(* Logix 5000 project; controller Transcat_L33ER vendor 1 type 14 code 107 rev 32.11; software revision 32.02 *)
// Upgraded CPLX to handle up to 32 EIP Nodes

TASK MainTask (continuous, watchdog 500 ms) : MainProgram

MODULES
   Local : vendor 1 type 14 code 107 (Compact 0, rev 32.11)
        TC_Remote_IO:5:O.0   // HOIST 2 BEACON RED
        TC_Remote_IO:5:O.1   // CV_101 - 3 Way Valve - Recyle / Process
        TC_Remote_IO:3:O.6   // HOIST 1 Beacon Red
        TC_Remote_IO:3:O.5   // HOIST 1 BEACON GREEN
        TC_Remote_IO:3:O.7   // Hoist 2 BEACON GREEN
        TC_Remote_IO:3:O   // HOIST 1 RED
      VFD9_Screener : PowerFlex 525-EENET (Ethernet 192.168.1.199, rev 5.1, Output RPI 20 ms)   // Screener Kaison
      GF201_Bentonite_Feeder : PowerFlex 525-EENET (Ethernet 192.168.1.195, rev 5.1, Output RPI 20 ms)   // Thayer Weigh Belt Feeder
      MX101_UpperHowesVFD : PowerFlex 525-EENET (Ethernet 192.168.1.191, rev 5.1, Output RPI 20 ms)   // VFD for Upper Howes Mixer
           MX101_UpperHowesVFD:I.Ready   // UpperHowes Drive Ready Status
           MX101_UpperHowesVFD:I.DriveStatus.1   // 1 = Running, 0 - Stopped
           MX101_UpperHowesVFD:I.DriveStatus.0   // 1 = Drive is Ready
           MX101_UpperHowesVFD:I.DriveStatus.4   // 1 = Accelerating
           MX101_UpperHowesVFD:I.DriveStatus.10   // 1 - parameter locked
           MX101_UpperHowesVFD:I.DriveStatus.8   // 1 = At Referecne Speed
           MX101_UpperHowesVFD:I.Faulted   // UpperHowes Drive Faulted
           MX101_UpperHowesVFD:I.DriveStatus.6   // not used
           MX101_UpperHowesVFD:I.DriveStatus.9   // 1 - Main Freq by Active Comms
           MX101_UpperHowesVFD:I.DriveStatus.3   // 1 = Rotating Forward
           MX101_UpperHowesVFD:I.DriveStatus.7   // 1= Faulted
           MX101_UpperHowesVFD:I.DriveStatus.2   // 1 = Forward, 0 = Reverse
           MX101_UpperHowesVFD:I.Active   // UpperHowes Drive Active
           MX101_UpperHowesVFD:I.DriveStatus.5   // 1= Decelerating
           MX101_UpperHowesVFD:O.Start   // Drive Start
           MX101_UpperHowesVFD:O.FreqCommand   // Input Hz into Source A: 0-60 Hz range
           MX101_UpperHowesVFD:O.Stop   // Drive Stop
      VF101_Medium_Feeder : PowerFlex 525-EENET (Ethernet 192.168.1.196, rev 5.1, Output RPI 20 ms)   // Medium Feeder
      MX201_LowerHowesVFD : PowerFlex 525-EENET (Ethernet 192.168.1.192, rev 5.1, Output RPI 20 ms)   // VFD for Lower Howes Mixer
           MX201_LowerHowesVFD:I.Ready   // LowerHowes Drive Ready Status
           MX201_LowerHowesVFD:I.Faulted   // LowerHowes Drive Faulted
           MX201_LowerHowesVFD:I.Active   // LowerHowes Drive Active
           MX201_LowerHowesVFD:O.Stop   // Drive Stop
      VF201_Small_Feeder_2 : PowerFlex 525-EENET (Ethernet 192.168.1.197, rev 5.1, Output RPI 20 ms)   // Acrison Small Feeder 2
      Anybus_ETH_SER : ETHERNET-MODULE (Ethernet 192.168.1.127, rev 1.1, Output RPI 50 ms)   // Anybus gateway from serial (Bronkhorst) to / from EIP (Ether/IP) - PLC
      SBC2000_1_Acrison : ETHERNET-MODULE (Ethernet 192.168.1.150, rev 1.1, Output RPI 250 ms)   // Acrison Drive 1 to control Small Feeder 1
           SBC2000_1_Acrison:I.Data   // Ethernet Input Array
           SBC2000_1_Acrison:I.Data[1]   // PV - Feedrate - kg/hr
           SBC2000_1_Acrison:I.Data[2]   // Totalizer 1 - kg
           SBC2000_1_Acrison:I.Data[4]   // Hopper Level - %
           SBC2000_1_Acrison:I.Data[0]   // SP-FeedRate - kg/hr
           SBC2000_1_Acrison:I.Data[3]   // OT - Motor Speed - %
           SBC2000_1_Acrison:O.Data[15]   // When Command_Bits is 1, machine is running.
      Thayer1_BS : ETHERNET-MODULE (Ethernet 192.168.1.140, rev 1.1, Output RPI 50 ms)   // Thayer 1 Weight Belt Feeder
      Thayer2_BS : ETHERNET-MODULE (Ethernet 192.168.1.160, rev 1.1, Output RPI 50 ms)   // Thayer 2 Weigh Belt Feeder
      XS26_VFD_Cabinet_Safety_Controller : XS26 SC26 SC10 (Ethernet 192.168.1.212, rev 2.1, StandardDataDriven RPI 100 ms)   // Banner XS26 Safety Controller with 3 expansion modules in VFD cabinet
           XS26_VFD_Cabinet_Safety_Controller:I1.Data[0].7   // MX101 VFD STO - OK
           XS26_VFD_Cabinet_Safety_Controller:I1.Data[1].0   // MX201 VFD STO - OK
      XS26_PLC_Safety_Controller : XS26 SC26 SC10 (Ethernet 192.168.1.211, rev 2.1, StandardDataDriven RPI 100 ms)   // XS26 Safety Controller in PLC cabinet
      TC_Remote_IO : 1734-AENT (Ethernet 192.168.1.190, rev 6.1, Output RPI 20 ms)
         TC_8Pt_Analog_Input : vendor 1 type 115 code 210 (PointIO 1, rev 3.1, Input RPI 80 ms)
         TC_8pt_DC_Input_Sink : 1734-IB8 (PointIO 2, rev 3.1)
         TC_8pt_Digital_Output_Sourced : 1734-OB8 (PointIO 3, rev 3.1)
          : 1734-OB8 (PointIO 5, rev 3.1)   // For Hoist Safety Beacon
         TC_4pt_Relay_Output : 1734-OW4 (PointIO 4, rev 3.1)
END_MODULES

TYPE Acrison_Feeder :   // Acrison Feeder Tags
STRUCT
   AutoMan : BOOL;   // On - Auto Control - follows AutoRun bit, Off - Manaul Control - follows Manual Run bit
   ManualRun : BOOL;   // On - Runs feeder in Manual, Off - Stops feeder in manual
   AutoRun : BOOL;   // On - Runs feeder in Auto Off - Stops feeder in Auto
   Interlock : BOOL;   // Interlock bit - if on - Feeder will not run
   Output : BOOL;   // On - Feeder runs, Off Feeder stops
   Int_Status : DINT;   // 32 Status bits from feeder
   SP_HMI : REAL;   // setpoint from HMI
   SP_READ : REAL;   // setpoint read back from controller
   Enable : BOOL;   // Enable logic to run feeder
   OT_Actual_Hz : REAL;   // The current output of the VFD in Hz
   FreqHz_Real : REAL;   // The command frequency of the drive in Hz
   CycleTime : TIMER;   // running time of current cycle
   CampTime : TIMER;   // running time of current campaign / batch
   TotalTime : TIMER;   // total time the device / motor has run since last reset
   OneShots : BOOL[32];   // 32 Booleans to hold one-shots assicated with this device
   TimeRunTarget : DINT;   // Target Amount of time in seconds to run the device
   StartDelay : TIMER;   // Delay before motor start
   StartDelayms : DINT;   // Start delay in milliseconds
   TimeRunStart : BOOL;   // Bit to start and run a timed run
   RPM : REAL;   // RPM of shaft
END_STRUCT
END_TYPE

TYPE BronkhorstFlowMeter :   // Read and write values for Bronkhorst Flow Meters
STRUCT
   SP_R : REAL;   // Set Point - FlowRate - Read - g/min - read from Flow Meter
   PV_R : REAL;   // Process Variable - FlowRate - Read - g/min
   OT_R : REAL;   // Output - PumpSpeed - Read - %
   TempC : REAL;   // Temperaure - Read - Deg C
   Density : REAL;   // Density - Read - g/liter
   Usertag : STRING;   // User Tag in Flow Meter - String
   FBNode : INT;   // Flow Bus Node # - Integer
   Model : STRING;   // Flow Meter Model #
   Serial : STRING;   // Flow Meter Serial #
   Capacity : REAL;   // Max Flow Rate of Flow Meter
   Enable : BOOL;   // Device enable bit
   AutoMan : BOOL;   // Select Auto / Manual Mode
   AutoRun : BOOL;   // On / Off in Auto Mode
   ManualRun : BOOL;   // On / Off- in Manual Mode
   Interlock : BOOL;   // Interlock Bit
   Output : BOOL;   // Output Bit for Device
   SP_HMI : REAL;   // Setpoint from HMI
   SP_W : REAL;   // Setpoint - flowrate g/min - write to Flow Meter from PLC
   Connected : BOOL;   // Is flow meter connecte to the flow bus network
   Alarm : BOOL;   // Alarm Bit - if on flow meter in ALarm Status
   Running : BOOL;   // the flow meter is running / dosing
   AlarmReset : BOOL;   // bit to toggle to reset alarm
   AlarmID : INT;   // Integer # that describes the type of Alarm
   ReadTime : INT;   // time in milliseconds to read the flow meter data
   DevPct : REAL;   // % deviation of process variable from setpoint
   CycleTime : TIMER;   // running time of current cycle
   CampTime : TIMER;   // running time of current campaign
   TotalTime : TIMER;   // total time the device / motor has run since last reset
   OneShots : BOOL[32];   // 32 Booleans to hold one-shots assicated with this device
   TimeRunTarget : DINT;   // Target Amount of time in seconds to run the device
   StartDelay : TIMER;   // Delay before motor start
   StartDelayms : DINT;   // Start delay in milliseconds
   TimeRunStart : BOOL;   // Bit to start and run a timed run
   Totalizer : REAL;   // Total dosed by flow meter since last reset
   TotalizerReset : BOOL;   // Bit to reset the totalizer (called a counter in Bronkhorst literature)
   TotalizerEnable : BOOL;   // Bit to turn the totalizer on / off
   HighPressureLimit_HMI : REAL;   // High Pressure Limit Real Value in psi from HMI
   HighPressureLimit_Int : DINT;   // High Pressure limit converted to Int * 100 so 40.0 real = 4000 Int value
   HighPressureTime : DINT;   // Presistance time for high pressure limit
   HighPressureTimer : TIMER;   // Timer to time how many consecutive seconds the line pressur can stay above the limit before interlockig the pump / flow meter system
   HighPressureInterlock : BOOL;   // The pump / flow meter dosign system is interlocked due to a high pressure event
   TotalResetCmd : BOOL;   // Total Reset Command from HMI
   TotalResetDone : BOOL;   // Gateway confirms totalizer is near zero
   TotalResetError : BOOL;   // Reset failed after the retry limit
   AlarmResetCmd : BOOL;   // PLC/HMI requests alarm reset
   AlarmResetDone : BOOL;   // Gateway confirms alarm reset
   AlarmResetError : BOOL;   // Alarm didn't clear / reset failed
   TotalResetAttempts : DINT;   // Total Reset Attempts
   CommOK : BOOL;   // Meter communications are healthy
   DataValid : BOOL;   // Current data is good and not stale
   DataStale : BOOL;   // Data is no longer considered current
   DataAgeMs : DINT;   // Milliseconds since last good meter data
END_STRUCT
END_TYPE

TYPE Device :   // this UDT will be the template for all equipment / devices - feeders, flow meters, others and will be set up for each device to be indexed and processed via indirect addressing
STRUCT
   SP_R : REAL;   // Set Point - FlowRate - Read - g/min - read from Flow Meter
   PV_R : REAL;   // Process Variable - FlowRate - Read - g/min
   OT_R : REAL;   // Output - PumpSpeed - Read - %
   TempC : REAL;   // Temperaure - Read - Deg C
   Density : REAL;   // Density - Read - g/liter
   Usertag : STRING;   // User Tag in Flow Meter - String
   FBNode : INT;   // Flow Bus Node # - Integer
   Model : STRING;   // Flow Meter Model #
   Serial : STRING;   // Flow Meter Serial #
   Capacity : REAL;   // Max Flow Rate of Flow Meter
   Enable : BOOL;   // Device enable bit
   AutoMan : BOOL;   // Select Auto / Manual Mode
   AutoRun : BOOL;   // On / Off in Auto Mode
   ManualRun : BOOL;   // On / Off- in Manual Mode
   Interlock : BOOL;   // Interlock Bit
   Output : BOOL;   // Output Bit for Device
   SP_HMI : REAL;   // Setpoint from HMI
   SP_W : REAL;   // Setpoint - flowrate g/min - write to Flow Meter from PLC
   Connected : BOOL;   // Is flow meter connecte to the flow bus network
   Alarm : BOOL;   // Alarm Bit - if on flow meter in ALarm Status
   Running : BOOL;   // the flow meter is running / dosing
   AlarmReset : BOOL;   // bit to toggle to reset alarm
   AlarmID : INT;   // Integer # that describes the type of Alarm
   ReadTime : INT;   // time in milliseconds to read the flow meter data
   DevPct : REAL;   // % deviation of process variable from setpoint
   CycleTime : TIMER;   // running time of current cycle
   CampTime : TIMER;   // running time of current campaign
   TotalTime : TIMER;   // total time the device / motor has run since last reset
   OneShots : BOOL[32];   // 32 Booleans to hold one-shots assicated with this device
   TimedRunTarget : DINT;   // Target Amount of time in seconds to run the device
   StartDelay : TIMER;   // Delay before motor start
   StartDelayms : DINT;   // Start delay in milliseconds
   TimeRunEnable : BOOL;   // Bit to enable / activate a timed (campaign timed) run
   Totalizer : REAL;   // Total dosed by flow meter since last reset
   TotalizerReset : BOOL;   // Bit to reset the totalizer (called a counter in Bronkhorst literature)
   TotalizerEnable : BOOL;   // Bit to turn the totalizer on / off
   TimedRunTargetms : DINT;   // Timed run target convered to ms for use in timers
   OutPutTest : BOOL;   // A bit to simulate output that does NOT control anything
   StartDelay_ST_Timer : FBD_TIMER;   // Start delay timer to use in stuctured text
   PermissivesAuto : BOOL;   // Bit to allow device to start in AUTO as long as all permissive conditions met
   PermissivesMan : BOOL;   // Bit to allow device to start in Manual as long as all permissive conditions met
   Error : REAL;   // % Error from SP (Positive Value = running above SP and vice versa)
   ErrorTimer : TIMER;   // Amont of consecutive seconds the Error is permitterd to be out of range (+/- x%) before triggering interlock
   ErrorLimit : REAL;   // + / - % error range the system can operate in
   HMI_ManualStart : BOOL;   // Button that requests device start in Manual
   HMI_ManualStop : BOOL;   // Button that requesets device stop in Manual
   RunRequest : BOOL;   // One Bit that sets device output in Auto or Manual
   AutoEnable : BOOL;   // A bit to enable a device to run in Auto with other devices in Auto
   HMI_AutoSelect : BOOL;   // Select auto mode for device
   HMI_ManualSelect : BOOL;   // Select manual mode for device
   AutoArmed : BOOL;   // Tells the system device is in auto, but will needd fresh reestart to start when transitioning from manual back to Auto
   HMI_DeviceReset : BOOL;   // A bit that will be used to clear all interlocks and faultss specific to one device
   HMI_ProcessReset : BOOL;   // Reset process wide stop when all other interlocks are cleared
END_STRUCT
END_TYPE

TYPE Howes_Mixer :   // Howes Mixer Tags
STRUCT
   AutoMan : BOOL;   // On - Auto Control - follows AutoRun bit, Off - Manaul Control - follows Manual Run bit
   ManualRun : BOOL;   // On - Runs feeder in Manual, Off - Stops feeder in manual
   AutoRun : BOOL;   // On - Runs feeder in Auto Off - Stops feeder in Auto
   Interlock : BOOL;   // Interlock bit - if on - Feeder will not run
   Output : BOOL;   // On - Feeder runs, Off Feeder stops
   Int_Status : DINT;   // 32 Status bits from feeder
   SP_HMI : REAL;   // setpoint from HMI
   SP_READ : REAL;   // setpoint read back from controller
   Enable : BOOL;   // Enable logic to run mixer
   FreqHz_Real : REAL;   // Frequency in Hz expressed as real #
   OT_Actual_Hz : REAL;   // The current output of the drive in Hz
   CycleTime : TIMER;   // currnet cycle run time
   CampTime : TIMER;   // current campaign run time
   TotalTime : TIMER;   // total run time since last reset
   OneShots : BOOL[32];   // 32 Booleans to hold one shots associated with this device
   TimeRunTarget : DINT;   // Target Amount of time in seconds to run the device
   TimeRunStart : BOOL;   // Bit to start and run a timed run
   StartDelay : TIMER;   // Delay before motor starts
   StartDelayms : DINT;   // Delay before motor starts in milliseconds
   RPM : REAL;   // RPM from speed sensor
END_STRUCT
END_TYPE

TYPE Thayer_WB_Feeder :   // Thayer WB Feeder Tags
STRUCT
   AutoMan : BOOL;   // On - Auto Control - follows AutoRun bit, Off - Manaul Control - follows Manual Run bit
   ManualRun : BOOL;   // On - Runs feeder in Manual, Off - Stops feeder in manual
   AutoRun : BOOL;   // On - Runs feeder in Auto Off - Stops feeder in Auto
   Interlock : BOOL;   // Interlock bit - if on - Feeder will not run
   Output : BOOL;   // On - Feeder runs, Off Feeder stops
   Int_Status : DINT;   // 32 Status bits from feeder
   SP_HMI : REAL;   // setpoint from HMI
   SP_READ : REAL;   // setpoint read back from controller
   Enable : BOOL;   // Enable logic to run feeder
   CycleTime : TIMER;   // current cycle run time
   CampTime : TIMER;   // current campaing run time
   TotalTime : TIMER;   // total run time since last reset
   OneShots : BOOL[32];   // 32 Booleans to hold one-shots assicated with this device
   TimeRunTarget : DINT;   // Target Amount of time in seconds to run the device - from recipe
   StartDelay : TIMER;   // Delay before starting motor / equipment
   StartDelayms : DINT;   // Start delay in milliseconds
   TimeRunStart : BOOL;   // Bit to start and run a timed run
END_STRUCT
END_TYPE

ADD_ON_INSTRUCTION HexASCII_to_REAL   (* revision 1.0 *)
// Converts 8-byte ASCII hex string (e.g. BF61F4AA) to REAL float
VAR_IN_OUT
   HexIn : SINT[8]; {required}   // "8 ASCII bytes (e.g. [66,70,54,49,70,52,65,65]) – passed by reference"
END_VAR
VAR_OUTPUT
   FloatOut : REAL; {access Read Only, required}   // Resulting floating-point value
   Error : BOOL; {access Read Only, required}   // 1 = invalid hex character or data
END_VAR
VAR
   Nibble : DINT; {access None}   // 4-bit value (0-15)
   TempByte : SINT; {access None}   // Current ASCII byte
   i : DINT; {access None}   // Loop Counter
   TempDINT : DINT; {access None}   // Temporary 32-bit hex value
END_VAR

ROUTINE Logic   (* structured text *)
// Converts 8-byte ASCII hex string (e.g. BF61F4AA) to REAL float
   // ================================================
   // HexASCII_to_REAL AOI Logic - Structured Text
   // Converts 8 ASCII hex bytes → IEEE 754 REAL
   // ================================================
   
   Error := 0;
   TempDINT := 0;
   
   // Parse each of the 8 hex characters
   FOR i := 0 TO 7 DO
       TempByte := HexIn[i];
   
       IF (TempByte >= 48) AND (TempByte <= 57) THEN          // '0' - '9'
           Nibble := TempByte - 48;
       ELSIF (TempByte >= 65) AND (TempByte <= 70) THEN       // 'A' - 'F' uppercase
           Nibble := TempByte - 55;
       ELSIF (TempByte >= 97) AND (TempByte <= 102) THEN      // 'a' - 'f' lowercase
           Nibble := TempByte - 87;
       ELSE
           Error := 1;          // Invalid character
           FloatOut := 0.0;
           EXIT;                // Break out of FOR loop early
       END_IF;
   
       // Build the 32-bit pattern (most-significant digit first)
       TempDINT := (TempDINT * 16) + Nibble;
   END_FOR;
   
   // Only perform COP if no error occurred
   IF NOT Error THEN
       COP(TempDINT, FloatOut, 1);
   END_IF;
END_ROUTINE
END_ADD_ON_INSTRUCTION

VAR_GLOBAL   (* controller tags *)
   AcrisonFeedRateSetPoint : MESSAGE;   // Message Command to Write to Feed Rate Set Point in Acrison from GF103.SP_HMI in kg/hr
        MessageParameters(ServiceCode := 16#0010, LocalElement := GF301.SP_HMI, ...)
   AcsiiToReal1 : HexASCII_to_REAL := (Error := 1);
   AllDevice1stScanDone : BOOL := 1;   // When this bit is set - all devices have been scanned once and bits reset
   AllDeviceEnable : BOOL := 1;   // A bit to enable or disable the running of all devices
   AllReset : BOOL;   // Bit to reset Auto/Man, AutoRun, RecipeRun, TimedRunEnable to 0 from PLC
   alwaysOFF : BOOL;
   AlwaysOFF2 : BOOL;
   AlwaysOn : BOOL := 1;
   AnyAutoRun : BOOL;   // Bit that in on if ANY device is placed into Auto run (to signal pre-start beed)
   AnyAutoRunFlag : BOOL;   // A flag that indicates if any device is in Auto Run (used with pre-start beep logic)
   AnyManRunFlag : BOOL;   // A flag that indicates if any device is in Manual Run (used with pre-start beep logic)
   AnyManualRun : BOOL;   // Bit that in on if ANY device is placed into manual run (to signal pre-start beed)
   AnyRun : BOOL := 1;   // Bit that is true if any Maunal Run or Auto Run bit is set
   AnyRunFlag : BOOL;   // A Flag to know if any device in already running in Auto or Manual
   Auto_Run_All_Interlock : BOOL := 1;   // Bit to interlock all devices running in Auto
   AutoActive : BOOL := 1;   // Auto mode active
   AutoStartOS : BOOL;   // Auto Start One-Shot
   AutoStopOS : BOOL;   // Auto Stop One-Shot
   BeaconBeepAlarm : BOOL;   // Beep Alarm
   BeaconBlueLight : ALIAS FOR TC_Remote_IO:3:O.3;   // Blue Beacon Light
   BeaconGreenLight : ALIAS FOR TC_Remote_IO:3:O.2;   // Green Beacon Light
   BeaconRedLight : ALIAS FOR TC_Remote_IO:3:O.0;   // Red Beacon Light
   BeaconYellowLight : ALIAS FOR TC_Remote_IO:3:O.1;   // Yellow Beacon Light
   Beep : BOOL;   // Bit to Activte Beacon Alarm
   BeepNew : ALIAS FOR TC_Remote_IO:3:O.4;
   Bronkhorst_In : REAL[50];   // Floating point data coming from EIP ready of 8 bytes and converted to 64 bit floaing point and stored here
   Bronkhorst_Out : REAL[50];   // Floating point data coming from PLC as 64 bit float and converted to to 8 bytes send to bronklhorst for setpoint and others
   bronkhorstReal : REAL[50] := ([49] := 0.7299429);   // data from Bonkhorst - convertred to real values
   BronkOutArr : DINT[3];   // 3 Outputs from Flow controllers 0 - 100% = 0 - 32000
   BronkRead4Int : DINT := -1897541825;   // Place to put the 4 values coming in from bronk via binary protocal
   BronkRead4SINT : SINT := 63;   // Place to put the 4 values coming in from bronk via binary protocal
   BronkReal : REAL := 1.5976925;   // Place to write 4 BYTES coming in from Par Pro Binary Protoal
   BronkRealInArr : REAL[100] := ([99] := -1.49e-43);
   BronkRealOutArr : DINT;
   ConversionError : BOOL := 1;
   ConvertedFloat : REAL;
   CV_101_Output : ALIAS FOR TC_Remote_IO:5:O.1;   // CV_101 - 3 Way Valve - Recyle / Process
   dataIndex : DINT := 340;   // Bronkhorst Data Index
   Device : Device[20] := ([0].SP_HMI := 10.6, [0].CycleTime.PRE := 288000000, [0].CycleTime.ACC := 3998, [0].CampTime.PRE := 288000000, [0].CampTime.ACC := 20003, [0].TotalTime.PRE := 288000000, [0].TotalTime.ACC := 35952700, [0].TimedRunTarget := 20, [0].StartDelay.PRE := 1000, [0].StartDelayms := 1, [0].TimedRunTargetms := 20000, [0].StartDelay_ST_Timer.TimerEnable := 1, [0].StartDelay_ST_Timer.PRE := 10000, [0].PermissivesAuto := 1, [0].PermissivesMan := 1, [0].ErrorTimer.PRE := 1000, [1].SP_HMI := 10.6, [1].CycleTime.PRE := 288000000, [1].CycleTime.ACC := 3999, [1].CampTime.PRE := 288000000, [1].CampTime.ACC := 20004, [1].TotalTime.PRE := 288000000, [1].TotalTime.ACC := 29849279, [1].TimedRunTarget := 20, [1].StartDelay.PRE := 1000, [1].StartDelayms := 1, [1].TimedRunTargetms := 20000, [1].PermissivesAuto := 1, [1].PermissivesMan := 1, [1].ErrorTimer.PRE := 60000, [2].CycleTime.PRE := 288000000, [2].CycleTime.ACC := 4371, [2].CampTime.PRE := 288000000, [2].CampTime.ACC := 5003, [2].TotalTime.PRE := 288000000, [2].TotalTime.ACC := 22497901, [2].TimedRunTarget := 5, [2].StartDelay.PRE := 1000, [2].StartDelayms := 1, [2].TimedRunTargetms := 5000, [2].PermissivesAuto := 1, [2].PermissivesMan := 1, [2].Error := -98.929855, [3].CycleTime.PRE := 288000000, [3].CycleTime.ACC := 4372, [3].CampTime.PRE := 288000000, [3].TotalTime.PRE := 288000000, [3].TotalTime.ACC := 115659048, [3].TimedRunTarget := 10, [3].StartDelay.PRE := 1000, [3].StartDelayms := 1, [3].TimedRunTargetms := 10000, [3].PermissivesAuto := 1, [3].PermissivesMan := 1, [3].Error := -100.0, [4].CycleTime.PRE := 288000000, [4].CycleTime.ACC := 9975, [4].CampTime.PRE := 288000000, [4].TotalTime.PRE := 288000000, [4].TotalTime.ACC := 1550491,
        [4].StartDelay.PRE := 1000, [4].StartDelayms := 1, [4].PermissivesAuto := 1, [4].PermissivesMan := 1, [5].CycleTime.PRE := 288000000, [5].CycleTime.ACC := 4976, [5].CampTime.PRE := 288000000, [5].CampTime.ACC := 39951, [5].TotalTime.PRE := 288000000, [5].TotalTime.ACC := 12762696, [5].TimedRunTarget := 120, [5].StartDelay.PRE := 1000, [5].StartDelayms := 1, [5].TimedRunTargetms := 120000, [5].PermissivesAuto := 1, [5].PermissivesMan := 1, [6].CycleTime.PRE := 288000000, [6].CycleTime.ACC := 2974, [6].CampTime.PRE := 288000000, [6].CampTime.ACC := 39952, [6].TotalTime.PRE := 288000000, [6].TotalTime.ACC := 6477554, [6].TimedRunTarget := 120, [6].StartDelay.PRE := 1000, [6].StartDelayms := 1, [6].TimedRunTargetms := 120000, [6].PermissivesAuto := 1, [6].PermissivesMan := 1, [7].AutoMan := 1, [7].SP_HMI := 150.0, [7].CycleTime.PRE := 288000000, [7].CycleTime.ACC := 7924, [7].CampTime.PRE := 288000000, [7].CampTime.ACC := 39951, [7].TotalTime.PRE := 288000000, [7].TotalTime.ACC := 44758778, [7].TimedRunTarget := 120, [7].StartDelay.PRE := 1000, [7].StartDelayms := 1, [7].TimedRunTargetms := 120000, [7].PermissivesAuto := 1, [7].PermissivesMan := 1, [7].Error := -13.912079, [7].ErrorTimer.PRE := 1000, [7].AutoEnable := 1, [8].AutoMan := 1, [8].CycleTime.PRE := 288000000, [8].CycleTime.ACC := 7923, [8].CampTime.PRE := 288000000, [8].CampTime.ACC := 39952, [8].TotalTime.PRE := 288000000, [8].TotalTime.ACC := 32949360, [8].TimedRunTarget := 120, [8].StartDelay.PRE := 1000, [8].StartDelayms := 1, [8].TimedRunTargetms := 120000, [8].PermissivesAuto := 1, [8].PermissivesMan := 1, [8].Error := -35.01083, [8].ErrorTimer.PRE := 1000,
        [9].CycleTime.PRE := 288000000, [9].CycleTime.ACC := 11271, [9].CampTime.PRE := 288000000, [9].CampTime.ACC := 39951, [9].TotalTime.PRE := 288000000, [9].TotalTime.ACC := 41567477, [9].TimedRunTarget := 120, [9].StartDelay.PRE := 1000, [9].StartDelayms := 1, [9].TimedRunTargetms := 120000, [9].PermissivesAuto := 1, [9].PermissivesMan := 1, [9].Error := 0.53758097, [9].ErrorTimer.PRE := 1000, [10].CycleTime.PRE := 288000000, [10].CampTime.PRE := 288000000, [10].TotalTime.PRE := 288000000, [10].OneShots[2] := 1, [11].CycleTime.ACC := 11, [11].CycleTime.DN := 1, [11].TotalTime.ACC := 7, [11].TotalTime.DN := 1, [11].StartDelay.PRE := 1000, [11].StartDelayms := 1, [11].PermissivesAuto := 1, [11].PermissivesMan := 1, [12].CycleTime.ACC := 3, [12].CycleTime.DN := 1, [12].TotalTime.ACC := 8, [12].TotalTime.DN := 1, [12].StartDelay.PRE := 1000, [12].StartDelayms := 1, [12].PermissivesAuto := 1, [12].PermissivesMan := 1, [13].CycleTime.ACC := 2, [13].CycleTime.DN := 1, [13].TotalTime.ACC := 8, [13].TotalTime.DN := 1, [13].StartDelay.PRE := 1000, [13].StartDelayms := 1, [13].PermissivesAuto := 1, [13].PermissivesMan := 1, [14].OneShots[0] := 1, [14].OneShots[1] := 1, [14].OneShots[3] := 1, [14].OneShots[4] := 1);
        [8]   // FT104 - Bronkhorst Water Dosing System
        [0]   // MX101 - Upper Howes Mixer
        [1]   // MX201 - Lower Howes Mixer
        [12]   // SC1_Screener
        [2]   // GF101 - Thayer1 WB Feeder
        [3]   // GF201 - Thayer2 WB Feeder
        [9]   // FT105 Bronkhorst Fragrance Dosing System
        [5]   // VF101 Medium Feeder - Acurate
        [4]   // GF301 Small Feeder - Acrison LIW
        [13]   // CV-101 - 3 way valve
        [10]   // not used
        [11]   // Auxillary Pump
        [7]   // FT103 - Bronkhorst Oil Dosing System
        [6]   // VF201 Small Feeder 2 - Acrison
   DINT_Temp : DINT;   // Place to hold Dint's durng transition to new PLC
   DiscreteTemp : BOOL;   // A temporay boolean to hold positions during PLC transer
   dNum : DINT := 4;   // The index of the current device being processed
   DoseCounter : COUNTER := (ACC := 522, CU := 1, DN := 1);   // Counts the # of doses since last reset
   DoseCounterReset_HMI : BOOL;   // HMI bit to reset the dose counter
   DoseStart : BOOL;   // Bit to start dosing sequence
   DoseStartOneShot : BOOL := 1;   // One shot to start dosing
   DoseStop : BOOL;   // Bit to stop dosing
   DoseStopOneShot : BOOL := 1;   // one shot to stop dosing
   DoseTarget : REAL := 27.9;   // Target dose amount
   FT103 : BronkhorstFlowMeter := (Usertag := 'FT-103', Model := 'M55-RGD-25-0-S', Serial := 'M22213015A', Capacity := 1000.00006, Enable := 1, SP_HMI := 338.0, ReadTime := 500, CycleTime.PRE := 288000000, CycleTime.ACC := 19487, CampTime.PRE := 28800000, CampTime.ACC := 10001, TotalTime.PRE := 999999999, TotalTime.ACC := 114629, TotalizerEnable := 1, HighPressureLimit_HMI := 45.0, HighPressureLimit_Int := 4500, HighPressureTime := 1, HighPressureTimer.PRE := 1000);
   FT103B : BronkhorstFlowMeter := (PV_R := 0.72383016, TempC := 25.967249, Density := 9999.0, Usertag := 'FT-103', FBNode := 13, Model := 'M55-RGD-25-0-S', Serial := 'M22213015A', Capacity := 1000.00006, SP_HMI := 300.0, Connected := 1, Alarm := 1, AlarmID := 40, ReadTime := 94, Totalizer := 68.69, TotalizerEnable := 1, HighPressureLimit_HMI := 10.0, HighPressureLimit_Int := 1000, HighPressureTime := 2, HighPressureTimer.PRE := 2000, AlarmResetDone := 1, CommOK := 1, DataValid := 1, DataAgeMs := 63);
   FT104 : BronkhorstFlowMeter := (Usertag := 'FT-104          ', Model := 'M55-RGD-25-0-S', Serial := 'M22213015C', Capacity := 10000.0, Enable := 1, SP_HMI := 100.0, ReadTime := 500, CycleTime.PRE := 288000000, CycleTime.ACC := 3248, CampTime.PRE := 28800000, CampTime.ACC := 10001, TotalTime.PRE := 999999999, TotalTime.ACC := 84417, StartDelay.PRE := 2000, StartDelayms := 2, TotalizerEnable := 1, HighPressureLimit_HMI := 20.0, HighPressureLimit_Int := 2000, HighPressureTime := 1, HighPressureTimer.PRE := 1000, HighPressureInterlock := 1);
   FT104B : BronkhorstFlowMeter := (PV_R := 71.97906, TempC := 26.005651, Density := 9998.999, Usertag := 'FT-104          ', FBNode := 14, Model := 'M55-RGD-25-0-S', Serial := 'M22213015C', Capacity := 10000.0, SP_HMI := 1000.0, Connected := 1, ReadTime := 143, Totalizer := 2156.6, TotalizerEnable := 1, HighPressureLimit_HMI := 3.0, HighPressureLimit_Int := 300, HighPressureTime := 1, HighPressureTimer.PRE := 1000, CommOK := 1, DataValid := 1, DataAgeMs := 77);
   FT105 : BronkhorstFlowMeter := (Usertag := 'FT-105          ', Model := 'M14-RGD-22-0-S', Serial := 'M20210127A', Capacity := 202.79999, Enable := 1, SP_HMI := 100.0, ReadTime := 500, CycleTime.PRE := 288000000, CycleTime.ACC := 11357, CampTime.PRE := 28800000, CampTime.ACC := 10001, TotalTime.PRE := 999999999, TotalTime.ACC := 55929, StartDelay.PRE := 4000, StartDelayms := 4, TotalizerEnable := 1, HighPressureLimit_HMI := 45.0, HighPressureLimit_Int := 4500, HighPressureTime := 1, HighPressureTimer.PRE := 1000);
   FT105B : BronkhorstFlowMeter := (PV_R := 0.20980434, TempC := 29.442924, Density := 1005.667, Usertag := 'FT-105          ', FBNode := 15, Model := 'M14-RGD-22-0-S', Serial := 'M20210127A', Capacity := 202.79999, SP_HMI := 150.0, Connected := 1, ReadTime := 47, Totalizer := 296.41, TotalizerEnable := 1, HighPressureLimit_HMI := 2.0, HighPressureLimit_Int := 200, HighPressureTime := 1, HighPressureTimer.PRE := 1000, AlarmResetError := 1, CommOK := 1, DataValid := 1, DataAgeMs := 61);
   GF101 : Thayer_WB_Feeder := (SP_HMI := 18.0, SP_READ := 18.0, Enable := 1, CycleTime.PRE := 288000000, CycleTime.ACC := 9195, CampTime.PRE := 28800000, CampTime.ACC := 10001, TotalTime.PRE := 999999999, TotalTime.ACC := 1761327, StartDelay.PRE := 2000, StartDelayms := 2);   // Thayer 1 Tags
   GF101_Alarm_ExcessDevSP : ALIAS FOR Thayer1_BS:I.Data[8].7;   // Thayer 1 (GF101) - Alarm - excessive deviation from SP
   GF101_LoadCell : ALIAS FOR Thayer1Data[15];   // Thayer 1 (GF101) load cell in lbs
   GF101_LoadCellTempF : ALIAS FOR Thayer1Data[16];   // Thayer 1 (GF101) load cell temperature in Deg F
   GF101_OutputPct : ALIAS FOR Thayer1Data[5];   // Thayer 1 (GF101) Output to motor in pct - raw
   GF101_RunningLoad : ALIAS FOR Thayer1Data[0];   // Thayer 1 (GF101) Running Load - current load on belt in lbs
   GF101_RunningRate : ALIAS FOR Thayer1Data[1];   // Thayer 1 (GF101) Running Rate - current PV displayed on the operator screen
   GF101_RunningSpeed : ALIAS FOR Thayer1Data[2];   // Thayer 1 (GF101) Running Soeed - current speed of the belt in ft/min?
   GF101_SetPoint : ALIAS FOR Thayer1Data[3];   // Thayer 1 (GF101) SetPoint - in lb/min
   GF101_Shutdown_ExcessDevSp : ALIAS FOR Thayer1_BS:I.Data[10].7;   // Thayer 1 (GF101) - Shutdown - excessive deviation from SP
   GF101_Status_AutoMan : ALIAS FOR Thayer1_BS:I.Data[0].1;   // Thayer 1 (GF101) - Auto / Manual Status - 1 = Auto 0 = Manual
   GF101_Status_Coasting : ALIAS FOR Thayer1_BS:I.Data[0].2;   // Thayer 1 (GF101) - Coasting to stop of shutdown - 1 = Coasting, 0 = Not coasting
   GF101_Status_EchoBack : ALIAS FOR Thayer1_BS:I.Data[0].13;   // Thayer 1 (GF101) - Echo back bit
   GF101_Status_HeartBeat : ALIAS FOR Thayer1_BS:I.Data[0].14;   // Thayer 1 (GF101) - HeartBeat - every 5 seconds
   GF101_Status_Interlocked : ALIAS FOR Thayer1_BS:I.Data[0].8;   // Thayer 1 (GF101) - Interlocked Bit - 1 = Interlocked 0 = Not Interlocked
   GF101_Status_RunStop : ALIAS FOR Thayer1_BS:I.Data[0].0;   // Thayer 1 (GF101) - Operating Status - 1 = Running 0 = Stopped
   GF101_Status_TachGT0 : ALIAS FOR Thayer1_BS:I.Data[0].9;   // Thayer 1 (GF101) - 1 = Tachometer > 0 0 = Tachometer = 0
   GF101_TachHz : ALIAS FOR Thayer1Data[14];   // Thayer 1 (GF101) Tachometer in Hz
   GF101_Totalizer1 : ALIAS FOR Thayer1Data[9];   // Thayer 1 (GF101) Totalizer 1 in lbs
   GF101_Totalizer2 : ALIAS FOR Thayer1Data[10];   // Thayer 1 (GF101) Totalizer 2 in lbs
   GF101_Write_Acknowledge : ALIAS FOR Thayer1_BS:O.Data[2].5;   // Thayer 1 (GF101) Acknowledge
   GF101_Write_AutoMan : ALIAS FOR Thayer1_BS:O.Data[0].1;   // Thayer 1 (GF101) Auto / Manual 1 = Auto 2 = Manual
   GF101_Write_RunStop : ALIAS FOR Thayer1_BS:O.Data[0].0;   // Thayer 1 (GF101) 1 = Run / 0 = off/stop
   GF101_Write_Total1Reset : ALIAS FOR Thayer1_BS:O.Data[2].1;   // Thayer 1 (GF101) Totalizer 1 reset
   GF101_Write_Total2Reset : ALIAS FOR Thayer1_BS:O.Data[2].2;   // Thayer 1 (GF101) Totalizer 2 reset
   GF101OutpuyPct1sec : ALIAS FOR Thayer1Data[6];   // Thayer 1 (GF101) Output to motor in pct - averaged over 1 sec
   GF201 : Thayer_WB_Feeder := (SP_HMI := 18.0, SP_READ := 18.0, Enable := 1, CycleTime.PRE := 288000000, CycleTime.ACC := 17126, CampTime.PRE := 28800000, CampTime.ACC := 10001, TotalTime.PRE := 999999999, TotalTime.ACC := 1645614, StartDelay.PRE := 2000, StartDelayms := 2);   // Thayer 2 Tags
   GF201_Alarm_ExcessiDevSP : ALIAS FOR Thayer2_BS:I.Data[8].7;   // Thayer 2 (GF201) - Alarm - excessive deviation from SP
   GF201_LoadCell : ALIAS FOR Thayer2Data[15];   // Thayer 2 (GF201) load cell in lbs
   GF201_LoadCellTempF : ALIAS FOR Thayer2Data[16];   // Thayer 2 (GF201) load cell temperature in Deg F
   GF201_OutputPct : ALIAS FOR Thayer2Data[5];   // Thayer 2 (GF201) Output to motor in pct - raw
   GF201_RunningLoad : ALIAS FOR Thayer2Data[0];   // Thayer 2 (GF201) Running Load - current load on belt in lbs
   GF201_RunningRate : ALIAS FOR Thayer2Data[1];   // Thayer 2 (GF201) Running Rate - current PV displayed on the operator screen
   GF201_RunningSpeed : ALIAS FOR Thayer2Data[2];   // Thayer 2 (GF201) Running Soeed - current speed of the belt in ft/min?
   GF201_SetPoint : ALIAS FOR Thayer2Data[3];   // Thayer 2 (GF201) SetPoint - in lb/min
   GF201_Shutdown_ExcessDevSP : ALIAS FOR Thayer2_BS:I.Data[10].7;   // Thayer 2 (GF201) - Shutdown - excessive deviation from SP
   GF201_Status_AutoMan : ALIAS FOR Thayer2_BS:I.Data[0].1;   // Thayer 2 (GF201) - Auto / Manual Status - 1 = Auto 0 = Manual
   GF201_Status_Coasting : ALIAS FOR Thayer2_BS:I.Data[0].2;   // Thayer 2 (GF201) - Coasting to stop of shutdown - 1 = Coasting, 0 = Not coasting
   GF201_Status_EchoBack : ALIAS FOR Thayer2_BS:I.Data[0].13;   // Thayer 2 (GF201) - Echo back bit
   GF201_Status_HeartBeat1 : ALIAS FOR Thayer2_BS:I.Data[0].14;   // Thayer 2 (GF201) - HeartBeat - every 5 seconds
   GF201_Status_Interlocked : ALIAS FOR Thayer2_BS:I.Data[0].8;   // Thayer 2 (GF201) - Interlocked Bit - 1 = Interlocked 0 = Not Interlocked
   GF201_Status_RunStop : ALIAS FOR Thayer2_BS:I.Data[0].0;   // Thayer 2 (GF201) - Operating Status - 1 = Running 0 = Stopped
   GF201_Status_TachGT0 : ALIAS FOR Thayer2_BS:I.Data[0].9;   // Thayer 2 (GF201) - 1 = Tachometer > 0 0 = Tachometer = 0
   GF201_TachHz : ALIAS FOR Thayer2Data[14];   // Thayer 2 (GF201) Tachometer in Hz
   GF201_Totalizer1 : ALIAS FOR Thayer2Data[9];   // Thayer 2 (GF201) Totalizer 1 in lbs
   GF201_Totalizer2 : ALIAS FOR Thayer2Data[10];   // Thayer 2 (GF201) Totalizer 2 in lbs
   GF201_Write_Acknowledge : ALIAS FOR Thayer2_BS:O.Data[2].5;   // Thayer 2 (GF201) Acknowledge
   GF201_Write_AutoMan : ALIAS FOR Thayer2_BS:O.Data[0].1;   // Thayer 2 (GF201) Auto / Manual 1 = Auto 2 = Manual
   GF201_Write_RunStop : ALIAS FOR Thayer2_BS:O.Data[0].0;   // Thayer 2 (GF201) 1 = Run / 0 = off/stop
   GF201_Write_Total1Reset : ALIAS FOR Thayer2_BS:O.Data[2].1;   // Thayer 2 (GF1201) Totalizer 1 reset
   GF201_Write_Total2Reset : ALIAS FOR Thayer2_BS:O.Data[2].2;   // Thayer 2 (GF201) Totalizer 2 reset
   GF201OutpuyPct1sec : ALIAS FOR Thayer2Data[6];   // Thayer 2 (GF201) Output to motor in pct - averaged over 1 sec
   GF301 : Acrison_Feeder := (Int_Status := 591992, SP_HMI := 10.0, Enable := 1, CycleTime.PRE := 288000000, CycleTime.ACC := 223848, CampTime.PRE := 28800000, CampTime.ACC := 10001, TotalTime.PRE := 999999999, TotalTime.ACC := 2086091, StartDelay.PRE := 2000, StartDelayms := 2);   // GF103 - Small Feeder 1
        .Int_Status.3   // SP Int-1 / Ext-0
        .Int_Status.11   // Alarm
        .Output   // GF103 - Acrison Small Feeder Run Bit
        .Int_Status.13   // Empty
        .Int_Status.4   // Mode - Grav-1 / Vol-0
        .Int_Status.5   // Batch-1 / Cont-0
        .Int_Status.17   // Deviation
        .Int_Status.14   // Overfill
        .Int_Status.15   // Acrilock
        .Int_Status.10   // Overfill / Empty
        .Int_Status.16   // No Scale
        .Int_Status.1   // Refil
        .Int_Status.2   // AutoRefill
        .Int_Status.7   // Bribble
        .Int_Status.0   // Run-1 / Stop-0
        .Int_Status.6   // Batch Complete
        .Int_Status   // 32 Bit Status Int
        .Int_Status.8   // High Level
        .Int_Status.12   // Message
        .Int_Status.9   // Low Level
   GF301_AlarmAck : BOOL;   // GF301 Alarm Ack Bit
   GF301_ClearCommands : BOOL;   // Bit to send clear command to GF301 command integer
   GF301_Command_Bits : INT;   // Command Word - Holds a value that gets written to Acrison SCB2000:I.Data[15] see Acrison Manual for which bits do what
        .1   // Refill Mode Man - 1 / Auto - 0
        .8   // Setpoint - Ext -1 / Int - 0
        .4   // Refill ON
        .6   // Alarm Ack
        .5   // Refill OFF
        .3   // Batch Abort
        .7   // Mode Vol - 1/ Grav - 0
        .0   // Run-1 / Stop-0
        .2   // Batch-1 / Cont-0
   GF301_IntStatus : DINT := 591992;   // 32 Bit Status INT for GF301
        .14   // Overfill
        .12   // Message
        .15   // Acrilok
        .9   // Low Level
        .16   // No Scale
        .0   // Run- 1/ Stop - 0
        .3   // Setpoint Int - 1 / Ext - 0
        .17   // Deviation
        .1   // Refil
        .2   // Auto Refill
        .4   // Mode Grav - 1 / Vol - 0
        .8   // High Level
        .11   // Alarm
        .13   // Empty
        .10   // Overfill / Empty
        .7   // Dribble
        .6   // Batch Complete
        .5   // Batch - 1 / Cont - 0
   GF301_OT : ALIAS FOR SBC2000_1_Acrison:I.Data[3];   // GF301 Ouput ot motor in %
   GF301_PV : ALIAS FOR SBC2000_1_Acrison:I.Data[1];   // GF301 PV - Process Variable
   GF301_SP_READ : ALIAS FOR SBC2000_1_Acrison:I.Data[0];   // GF301 Set point read back from Acrison - kg/min
   GF301_TOTAL : ALIAS FOR SBC2000_1_Acrison:I.Data[2];   // GF301 Totalizer in KG
   GreenFlashingOff : TIMER := (PRE := 500);
   GreenFlashingOn : TIMER := (PRE := 500);
   HertzSetting : ALIAS FOR MX101_UpperHowesVFD:O.FreqCommand.0;   // UserHzSetting
   HMI_AllReset : BOOL;   // Bit to reset Auto/Man, AutoRun, RecipeRun, TimedRunEnable to 0 from HMI
   HMI_AutoStart : BOOL;   // Starts all devices in AUTO
   HMI_AutoStop : BOOL;   // Stops all devices in AUTO
   HMI_RecipeStart : BOOL;   // Bit to start and stop recipe from HMI
   InitCount : INT := 10;   // Counter to cycle through each device on start-up and reset AutoMan, AutoRun, ManualRun bits
   MSG_FROM_SLC500 : INT[10] := ([1] := 2500, [2] := 200, [3] := 300, [4] := 400, [5] := 500, [6] := 16, [7] := 17, [8] := 18, [9] := 19); {produced}
   MX101 : Howes_Mixer := (SP_HMI := 20.0, Enable := 1, FreqHz_Real := 6.67, CycleTime.PRE := 288000000, CycleTime.ACC := 4243, CampTime.PRE := 28800000, CampTime.ACC := 10001, TotalTime.PRE := 999999999, TotalTime.ACC := 1803981, TimeRunTarget := 10000, StartDelay.PRE := 2000, StartDelayms := 2, RPM := -0.12);
   MX101_RPM_RAW : ALIAS FOR Test_Hold;   // Raw (unscaled) RMS reading from MX101 speed sensor - RPM * 100 (range 0 - 200 RPM)
   MX101_Speed_Hold : DINT := 100;   // Constant Value for MX101 RPM meter - till Actual signal comes back from 4-20mA from sensor
   MX201 : Howes_Mixer := (AutoMan := 1, SP_HMI := 20.0, Enable := 1, FreqHz_Real := 6.67, CycleTime.PRE := 28800000, CycleTime.ACC := 117513, CampTime.PRE := 28800000, CampTime.ACC := 10001, TotalTime.PRE := 999999999, TotalTime.ACC := 1030054, TimeRunTarget := 10000, StartDelay.PRE := 2000, StartDelayms := 2, RPM := -0.08);
   MX201_RPM_RAW : ALIAS FOR Test_Hold;   // Raw (unscaled) RMS reading from MX201 speed sensor - RPM * 100 (range 0 - 200 RPM)
   MX201_Speed_Hold : DINT := 100;   // Constant Value for MX201 RPM meter - till Actual signal comes back from 4-20mA from sensor
   NewDataToggle : BOOL := 1;
   OldDeviceLogicEnable : BOOL;   // Enable old device logic
   PowerOffThayer1 : BOOL;
   PowerOnThayer1 : BOOL;
   PT103_HP_Interlock : BOOL;
   PT103_PV_RAW : ALIAS FOR TC_Remote_IO:1:I.Ch0Data;   // Raw (unscaled) pressure reading from PT103 - PSI * 100 (range 0 - 108 PSI)
   PT104_PV_RAW : ALIAS FOR TC_Remote_IO:1:I.Ch1Data;   // Raw (unscaled) pressure reading from PT104 - PSI * 100 (range 0 - 108 PSI)
   PT105_PV_RAW : ALIAS FOR TC_Remote_IO:1:I.Ch2Data;   // Raw (unscaled) pressure reading from PT105 - PSI * 100 (range 0 - 108 PSI)
   RandomFloat : REAL[20] := ([0] := 324.0, [1] := 13449296.0, [2] := 20.713356, [3] := 16.079597, [4] := 74.3938, [5] := 86.28061, [6] := 69.73996, [7] := 47.361, [8] := 43.876316, [9] := 89.62069, [10] := 12.1234);
   RandomSeed : DINT := 258;
   RandomTimer : TIMER := (PRE := 1000, ACC := 259, EN := 1, TT := 1);
   RealToBronkHorst : REAL[50];
        [0]   // Setpoint for FT103
        [1]   // Setpoint for FT104
        [2]   // Setpoint for FT105
   RecipeStart : BOOL;   // Bit to start and stop a recipe execution from PLC logic
   resultIndex : DINT := 47;   // Bronkhorst Real Result Index
   rms : BOOL;
   StartBeepTimer : TIMER := (PRE := 2500);   // Timer to sound the beep alarm before starting a device
   TempHexIn : SINT[8];   // Place to copy 8 SINT for proessing by AOI
   TempReal1 : REAL;
   Test_Hold : DINT;   // Place for RPM and Pressure sensors to Alias for while the AI's are not available
   TestBit1 : BOOL;   // Just a test bit - does not do anything
   testFloat : REAL;   // temp result for AsciiHex to real conversion
   Thayer1_SP : REAL := 20.0;
   Thayer1Ackn_SilenceRequest : BOOL;
   Thayer1Automatic : BOOL;
   Thayer1Data : REAL[40] := ([0] := -0.002456665, [1] := 3.3809e-41, [3] := 18.0, [4] := 2.0, [9] := 71.0, [10] := 1681.3524, [11] := 9.0565e-41, [15] := -0.0022277832, [16] := 70.35353, [17] := 8.7243e-41, [19] := -0.002456665);
        [2]   // Running Speed - belt speed in ft / min
        [1]   // Running Rate - Process variable in lb/min
        [7]   // not used
        [9]   // Totalizer 1
        [0]   // Running Load - load cell reading in lbs
        [14]   // Tachometer - Hz
        [8]   // not used
        [6]   // Drive Output in % (1 sec time averaged)
        [4]   // Ratio Setpoint - not used
        [5]   // Drive Output in %
        [12]   // take away belt load - not used
        [13]   // Take away belt rate - not used
        [10]   // Totalizer 2
        [16]   // Load Cell Temperatue - Deg F
        [17]   // Auto Zero error log in %
        [11]   // take a way totalizer - not used
        [15]   // Load Cell reading lbs.
        [3]   // SetPoint - in lb/min
   Thayer1PowerOn : BOOL;
   Thayer1ResetTotalizers : BOOL;
   Thayer1SetPoint : REAL[1];
   Thayer1SpeedControl : REAL := 20.0;
   Thayer2_SP : REAL := 20.0;
   Thayer2Automatic : BOOL;
   Thayer2Data : REAL[40] := ([0] := 2.75, [1] := 5.568e-41, [3] := 18.0, [9] := 71.0, [10] := 1734.9081, [11] := 7.929e-41, [15] := 2.75, [16] := 70.803085, [17] := 1.6071e-41, [19] := 2.75);
   Thayer2PowerOn : BOOL;
   Thayer2ResetTotal1_HMI : BOOL;   // Bit to reset Thayer2 - totalizer 1 from HMI
   Thayer2ResetTotalizers : BOOL;
   Thayer2SpeedControl : REAL := 20.0;
   TotalRestOneShot : BOOL;   // one shot for total reset
   UHStartOneShot : BOOL;
   UHStopOneShot : BOOL;
   UpHowesHMIRun : BOOL;
   UpHowesHMIStop : BOOL;
   UpHowesSpeedHMI : INT;
   UpperHowesSpeed : INT := 2500;
   UpperHowesStart : BOOL;
   UpperHowesStop : BOOL;
   UserBit1 : BOOL;   // user controlled bit for testing
   VF101 : Acrison_Feeder := (SP_HMI := 5.0, Enable := 1, FreqHz_Real := 3.0, CycleTime.PRE := 288000000, CycleTime.ACC := 7359, CampTime.PRE := 28800000, CampTime.ACC := 10001, TotalTime.PRE := 999999999, TotalTime.ACC := 1720239, StartDelay.PRE := 5000, StartDelayms := 5);   // Medium Feeder Tags
   VF201 : Acrison_Feeder := (SP_HMI := 5.0, Enable := 1, FreqHz_Real := 3.0, CycleTime.PRE := 288000000, CycleTime.ACC := 13534, CampTime.PRE := 28800000, CampTime.ACC := 10001, TotalTime.PRE := 999999999, TotalTime.ACC := 1964985, StartDelay.PRE := 5000, StartDelayms := 5);   // Small Feeder 2 Tags
   VFD_Panel_Safety_Any_Input_Fault : ALIAS FOR XS26_VFD_Cabinet_Safety_Controller:I1.Data[0].1;
   VFD_Panel_Safety_Any_Output_Fault : ALIAS FOR XS26_VFD_Cabinet_Safety_Controller:I1.Data[0].2;
   VFD_Panel_Safety_GF201_VF101_STO_OK : ALIAS FOR XS26_VFD_Cabinet_Safety_Controller:I1.Data[1].1;
   VFD_Panel_Safety_Hoist_1_Cart_OK : ALIAS FOR XS26_VFD_Cabinet_Safety_Controller:I1.Data[2].2;   // HOIST 1 Cart Sensor
   VFD_Panel_Safety_Hoist_1_K1_Disabled : ALIAS FOR XS26_VFD_Cabinet_Safety_Controller:I1.Data[2].4;
   VFD_Panel_Safety_Hoist_1_K2_Disabled : ALIAS FOR XS26_VFD_Cabinet_Safety_Controller:I1.Data[2].5;
   VFD_Panel_Safety_Hoist_1_OK : ALIAS FOR XS26_VFD_Cabinet_Safety_Controller:I1.Data[1].2;
   VFD_Panel_Safety_Hoist_2_Cart_OK : ALIAS FOR XS26_VFD_Cabinet_Safety_Controller:I1.Data[2].3;   // HOIST 2 Cart Sensor
   VFD_Panel_Safety_Hoist_2_K3_Disabled : ALIAS FOR XS26_VFD_Cabinet_Safety_Controller:I1.Data[2].6;
   VFD_Panel_Safety_Hoist_2_K4_Disabled : ALIAS FOR XS26_VFD_Cabinet_Safety_Controller:I1.Data[2].7;
   VFD_Panel_Safety_Hoist_2_OK : ALIAS FOR XS26_VFD_Cabinet_Safety_Controller:I1.Data[1].4;
   VFD_Panel_Safety_MX1012_Lid_Ok : ALIAS FOR XS26_VFD_Cabinet_Safety_Controller:I1.Data[2].1;
   VFD_Panel_Safety_MX101_Lid_Ok : ALIAS FOR XS26_VFD_Cabinet_Safety_Controller:I1.Data[2].0;
   VFD_Panel_Safety_MX101_MX201_STO_OK : ALIAS FOR XS26_VFD_Cabinet_Safety_Controller:I1.Data[0].7;
   VFD_Panel_Safety_Panel_Etop_OK : ALIAS FOR XS26_VFD_Cabinet_Safety_Controller:I1.Data[1].6;
   VFD_Panel_Safety_Remote_Estops_OK : ALIAS FOR XS26_VFD_Cabinet_Safety_Controller:I1.Data[1].7;
   VFD_Panel_Safety_SC_1_GF301_STO_OK : ALIAS FOR XS26_VFD_Cabinet_Safety_Controller:I1.Data[1].3;
   VFD_Panel_Safety_System_LockOut : ALIAS FOR XS26_VFD_Cabinet_Safety_Controller:I1.Data[0].0;
   VFD_Panel_Safety_VF201_GF101_STO_OK : ALIAS FOR XS26_VFD_Cabinet_Safety_Controller:I1.Data[1].0;
   YellowFlashOff : TIMER := (PRE := 500);
   YellowFlashOn : TIMER := (PRE := 500);
   ZS101_RPM_Speed_UpperHowes : ALIAS FOR TC_Remote_IO:1:I.Ch3Data;   // Upper Howes Zero Speed Sensor RPM
   ZS102_RPM_Speed_LowerHowes : ALIAS FOR TC_Remote_IO:1:I.Ch4Data;   // Lower Howes Zero Speed Sensor RPM
END_VAR

PROGRAM MainProgram   (* main routine MainRoutine *)
VAR
   AcrisonSpeedControl : REAL := 1.0;
   AcrisonSpeedControl2 : REAL := 15.0;
   HertzInput : INT := 20;
   Int_Status : DINT := 540252;
   LowerHowesSpeedSensor : REAL := -74.971405;
   MX101_Clr_VFd_Faults : BOOL;   // Bit to clear VFD faults
   PowerOffACrison : BOOL := 1;
   PowerOnAcrison : BOOL;
   SCL_01 : SCALE := (In := -21.0, InRawMax := 16384.0, InRawMin := 3271.0, InEUMax := 300.0, Out := -75.314575, MinAlarm := 1);
   SCL_02 : SCALE := (In := -6.0, InRawMax := 16384.0, InRawMin := 3271.0, InEUMax := 300.0, Out := -74.971405, MinAlarm := 1);
   SpeedSensorUpperHowesSpeed : REAL := -75.314575;
   T1 : TIMER := (PRE := 10000);
   T2 : TIMER := (PRE := 10000, ACC := 10000, EN := 1, DN := 1);
END_VAR

ROUTINE _00_MX101_UpperHowesMixer   (* ladder *)
// Upper Howes Mixer Specific (non Iteration) Control Logic
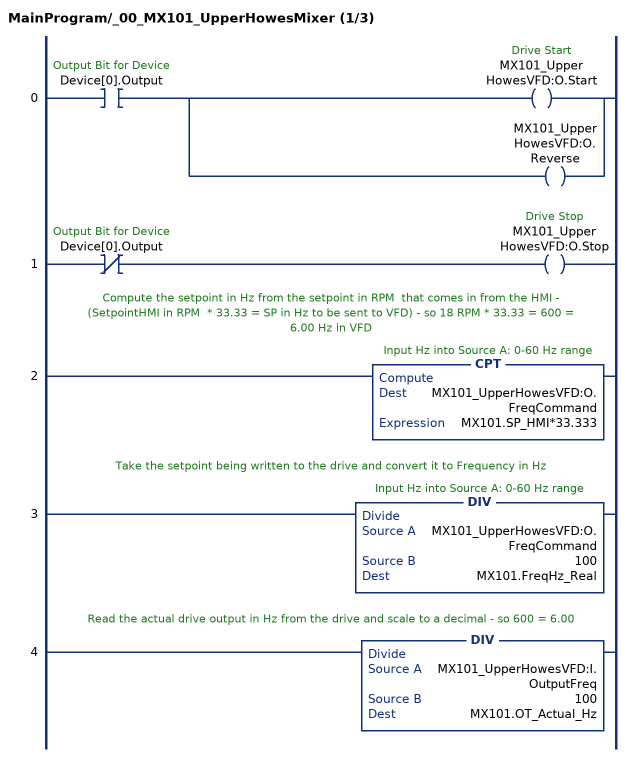
   0: XIC(Device[0].Output)[OTE(MX101_UpperHowesVFD:O.Start) ,OTE(MX101_UpperHowesVFD:O.Reverse) ];
   1: XIO(Device[0].Output)OTE(MX101_UpperHowesVFD:O.Stop);
   // Compute the setpoint in Hz from the setpoint in RPM  that comes in from the HMI - (SetpointHMI in RPM  * 33.33 = SP in Hz to be sent to VFD) - so 18 RPM * 33.33 = 600 = 6.00 Hz in VFD
   2: CPT(MX101_UpperHowesVFD:O.FreqCommand,MX101.SP_HMI*33.333);
   // Take the setpoint being written to the drive and convert it to Frequency in Hz
   3: DIV(MX101_UpperHowesVFD:O.FreqCommand,100,MX101.FreqHz_Real);
   // Read the actual drive output in Hz from the drive and scale to a decimal - so 600 = 6.00
   4: DIV(MX101_UpperHowesVFD:I.OutputFreq,100,MX101.OT_Actual_Hz);
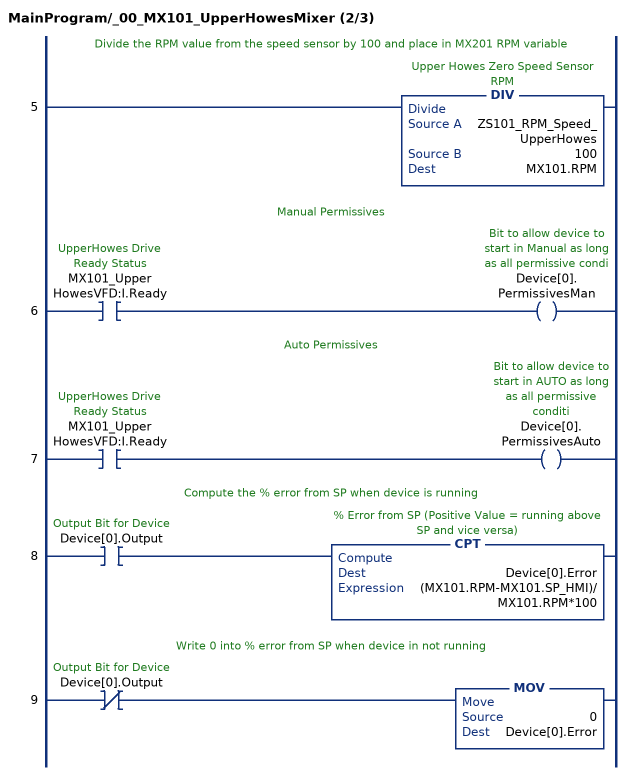
   // Divide the RPM value from the speed sensor by 100 and place in MX201 RPM variable
   5: DIV(ZS101_RPM_Speed_UpperHowes,100,MX101.RPM);
   // Manual Permissives
   6: XIC(MX101_UpperHowesVFD:I.Ready)OTE(Device[0].PermissivesMan);
   // Auto Permissives
   7: XIC(MX101_UpperHowesVFD:I.Ready)OTE(Device[0].PermissivesAuto);
   // Compute the % error from SP when device is running
   8: XIC(Device[0].Output)CPT(Device[0].Error,(MX101.RPM-MX101.SP_HMI)/MX101.RPM*100);
   // Write 0 into % error from SP when device in not running
   9: XIO(Device[0].Output)MOV(0,Device[0].Error);
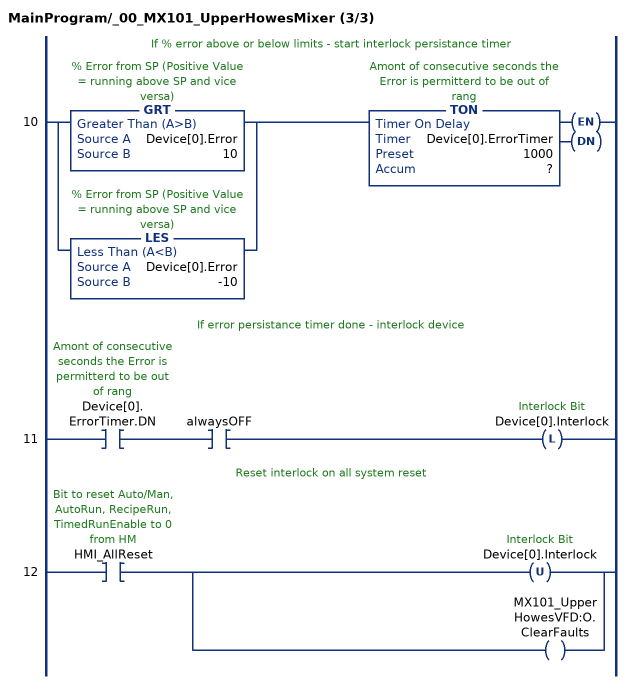
   // If % error above or below limits - start interlock persistance timer
   10: [GRT(Device[0].Error,10) ,LES(Device[0].Error,-10) ]TON(Device[0].ErrorTimer,?,?);
   // If error persistance timer done - interlock device
   11: XIC(Device[0].ErrorTimer.DN)XIC(alwaysOFF)OTL(Device[0].Interlock);
   // Reset interlock on all system reset
   12: XIC(HMI_AllReset)[OTU(Device[0].Interlock) ,OTE(MX101_UpperHowesVFD:O.ClearFaults) ];
END_ROUTINE

ROUTINE _01_MX201_LowerHowesMixer   (* ladder *)
// Lower Howes Mixer Control Logic not associated with Device Iteration Logic
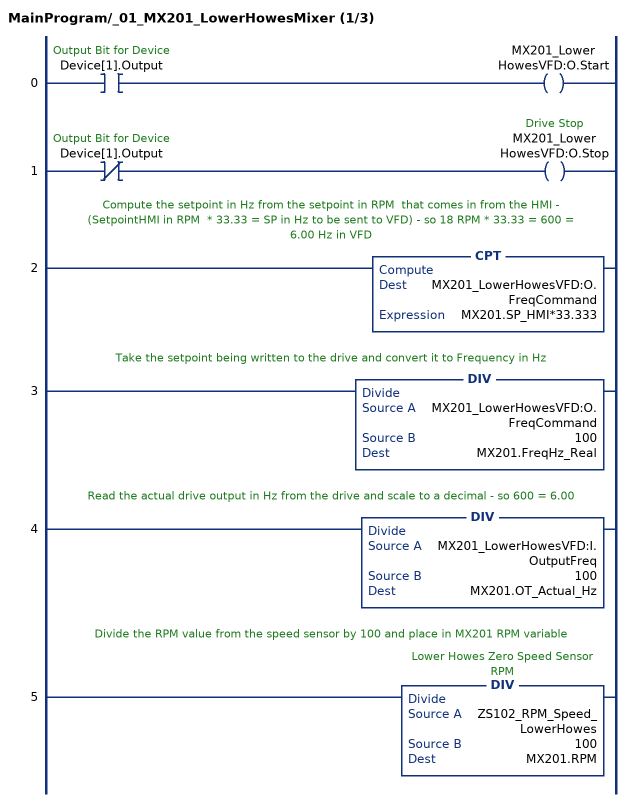
   0: XIC(Device[1].Output)OTE(MX201_LowerHowesVFD:O.Start);
   1: XIO(Device[1].Output)OTE(MX201_LowerHowesVFD:O.Stop);
   // Compute the setpoint in Hz from the setpoint in RPM  that comes in from the HMI - (SetpointHMI in RPM  * 33.33 = SP in Hz to be sent to VFD) - so 18 RPM * 33.33 = 600 = 6.00 Hz in VFD
   2: CPT(MX201_LowerHowesVFD:O.FreqCommand,MX201.SP_HMI*33.333);
   // Take the setpoint being written to the drive and convert it to Frequency in Hz
   3: DIV(MX201_LowerHowesVFD:O.FreqCommand,100,MX201.FreqHz_Real);
   // Read the actual drive output in Hz from the drive and scale to a decimal - so 600 = 6.00
   4: DIV(MX201_LowerHowesVFD:I.OutputFreq,100,MX201.OT_Actual_Hz);
   // Divide the RPM value from the speed sensor by 100 and place in MX201 RPM variable
   5: DIV(ZS102_RPM_Speed_LowerHowes,100,MX201.RPM);
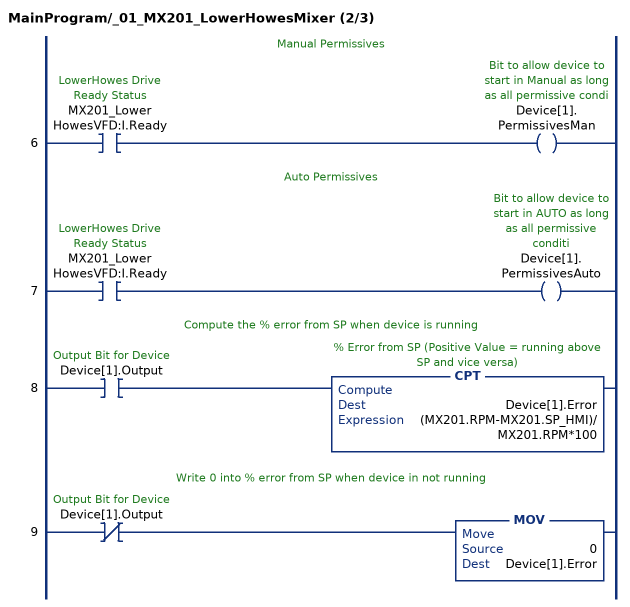
   // Manual Permissives
   6: XIC(MX201_LowerHowesVFD:I.Ready)OTE(Device[1].PermissivesMan);
   // Auto Permissives
   7: XIC(MX201_LowerHowesVFD:I.Ready)OTE(Device[1].PermissivesAuto);
   // Compute the % error from SP when device is running
   8: XIC(Device[1].Output)CPT(Device[1].Error,(MX201.RPM-MX201.SP_HMI)/MX201.RPM*100);
   // Write 0 into % error from SP when device in not running
   9: XIO(Device[1].Output)MOV(0,Device[1].Error);
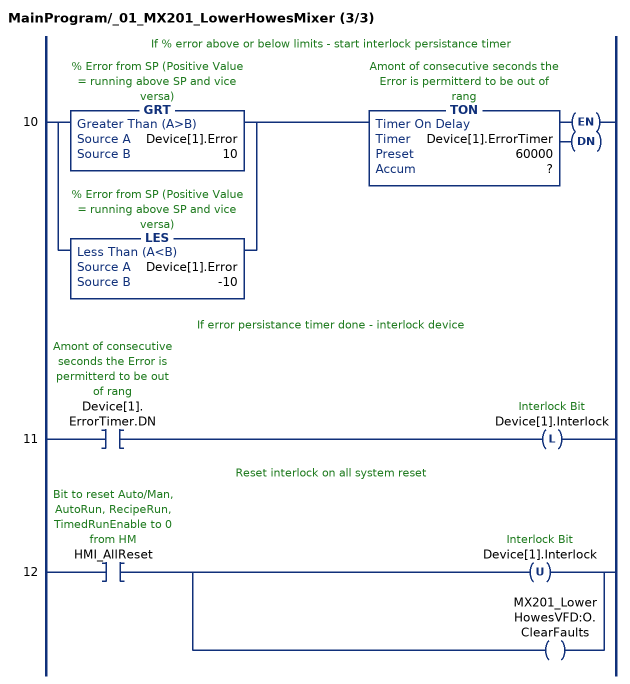
   // If % error above or below limits - start interlock persistance timer
   10: [GRT(Device[1].Error,10) ,LES(Device[1].Error,-10) ]TON(Device[1].ErrorTimer,?,?);
   // If error persistance timer done - interlock device
   11: XIC(Device[1].ErrorTimer.DN)OTL(Device[1].Interlock);
   // Reset interlock on all system reset
   12: XIC(HMI_AllReset)[OTU(Device[1].Interlock) ,OTE(MX201_LowerHowesVFD:O.ClearFaults) ];
END_ROUTINE

ROUTINE _02_GF101_Thayer1_WB_Feeder   (* ladder *)
// Thayer1 WB Feeder Control Logic (Old Limestone Feeder) - not associated with Device Iteration Logic
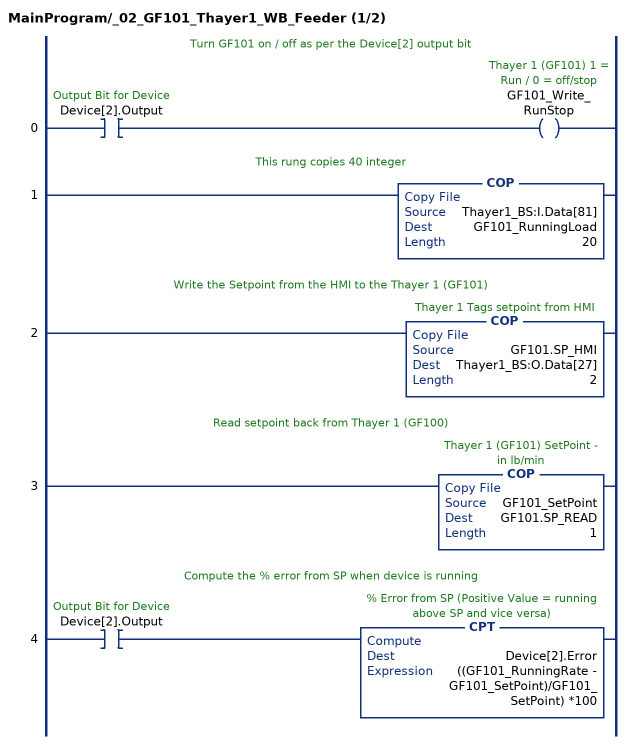
   // Turn GF101 on / off as per the Device[2] output bit
   0: XIC(Device[2].Output)OTE(GF101_Write_RunStop);
   // This rung copies 40 integer
   1: COP(Thayer1_BS:I.Data[81],GF101_RunningLoad,20);
   // Write the Setpoint from the HMI to the Thayer 1 (GF101)
   2: COP(GF101.SP_HMI,Thayer1_BS:O.Data[27],2);
   // Read setpoint back from Thayer 1 (GF100)
   3: COP(GF101_SetPoint,GF101.SP_READ,1);
   // Compute the % error from SP when device is running
   4: XIC(Device[2].Output)CPT(Device[2].Error,((GF101_RunningRate - GF101_SetPoint)/GF101_SetPoint) *100);
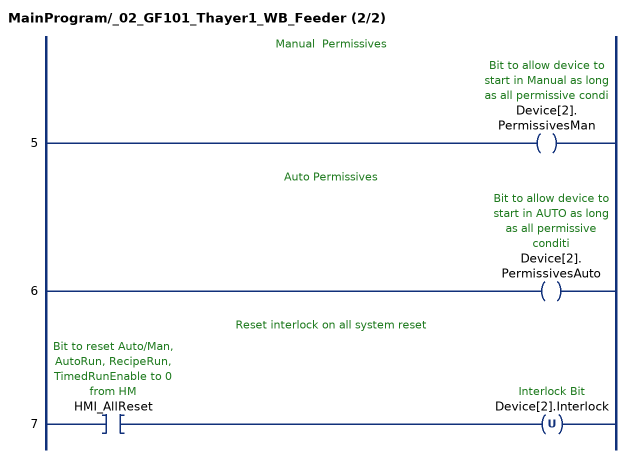
   // Manual  Permissives
   5: OTE(Device[2].PermissivesMan);
   // Auto Permissives
   6: OTE(Device[2].PermissivesAuto);
   // Reset interlock on all system reset
   7: XIC(HMI_AllReset)OTU(Device[2].Interlock);
END_ROUTINE

ROUTINE _03_GF201_Thayer2_WB_Feeder   (* ladder *)
// Thayer2 WB Feeder Control Logic (Old - Bentonite Feeder) not associated with Device Iteration Logic
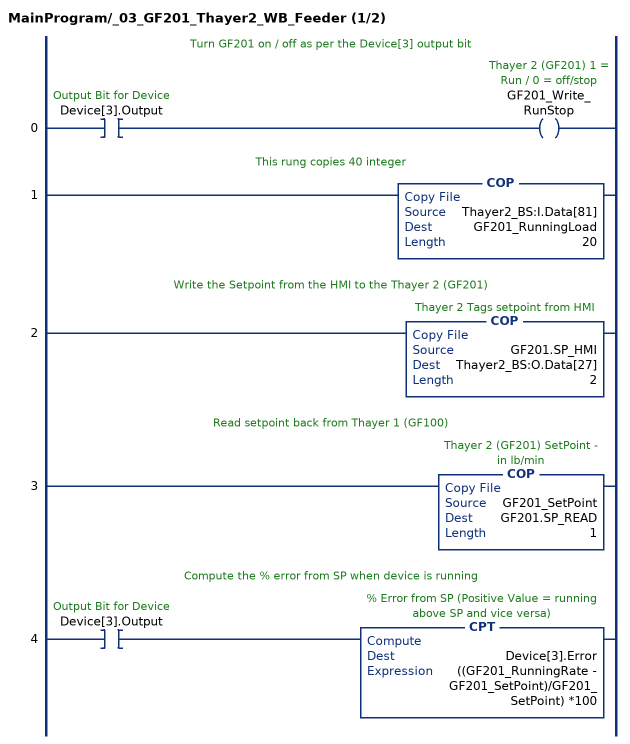
   // Turn GF201 on / off as per the Device[3] output bit
   0: XIC(Device[3].Output)OTE(GF201_Write_RunStop);
   // This rung copies 40 integer
   1: COP(Thayer2_BS:I.Data[81],GF201_RunningLoad,20);
   // Write the Setpoint from the HMI to the Thayer 2 (GF201)
   2: COP(GF201.SP_HMI,Thayer2_BS:O.Data[27],2);
   // Read setpoint back from Thayer 1 (GF100)
   3: COP(GF201_SetPoint,GF201.SP_READ,1);
   // Compute the % error from SP when device is running
   4: XIC(Device[3].Output)CPT(Device[3].Error,((GF201_RunningRate - GF201_SetPoint)/GF201_SetPoint) *100);
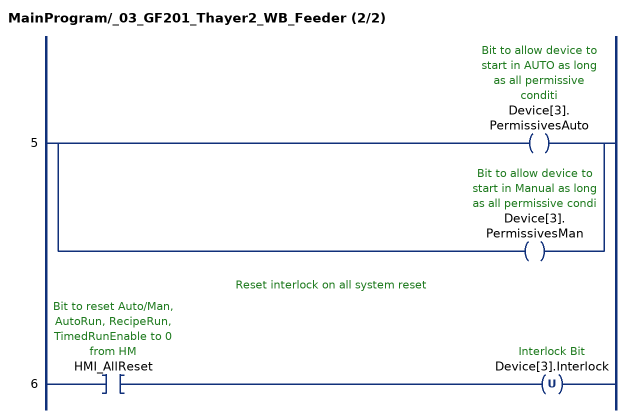
   5: [OTE(Device[3].PermissivesAuto) ,OTE(Device[3].PermissivesMan) ];
   // Reset interlock on all system reset
   6: XIC(HMI_AllReset)OTU(Device[3].Interlock);
END_ROUTINE

ROUTINE _04_GF301_Small_Feeder_AcrisonLIW   (* ladder *)
// Small Feeder 1 Control via Acrison Drive SBC 2000 - not associated with Device Iteration Logic
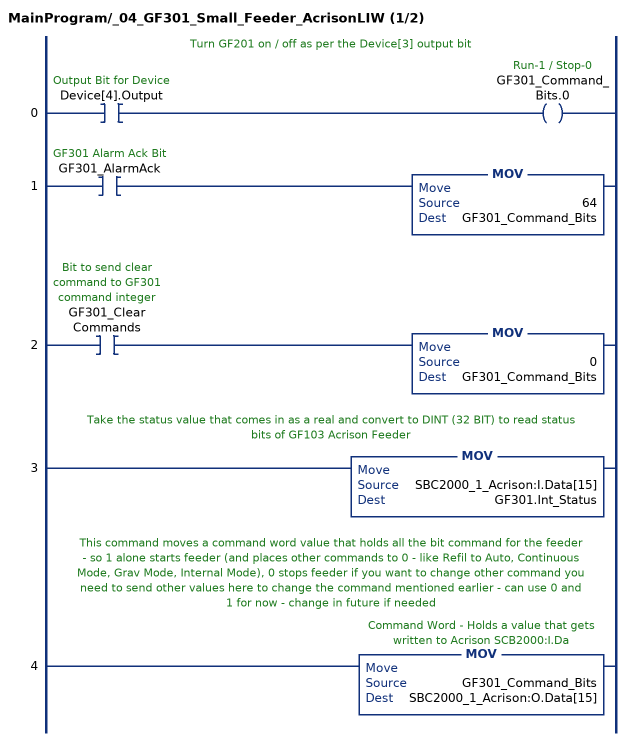
   // Turn GF201 on / off as per the Device[3] output bit
   0: XIC(Device[4].Output)OTE(GF301_Command_Bits.0);
   1: XIC(GF301_AlarmAck)MOV(64,GF301_Command_Bits);
   2: XIC(GF301_ClearCommands)MOV(0,GF301_Command_Bits);
   // Take the status value that comes in as a real and convert to DINT (32 BIT) to read status bits of GF103 Acrison Feeder
   3: MOV(SBC2000_1_Acrison:I.Data[15],GF301.Int_Status);
   // This command moves a command word value that holds all the bit command for the feeder - so 1 alone starts feeder (and places other commands to 0 - like Refil to Auto, Continuous Mode, Grav Mode, Internal Mode), 0 stops feeder if you want to change other command you need to send other values here to change the command mentioned earlier - can use 0 and 1 for now - change in future if needed
   4: MOV(GF301_Command_Bits,SBC2000_1_Acrison:O.Data[15]);
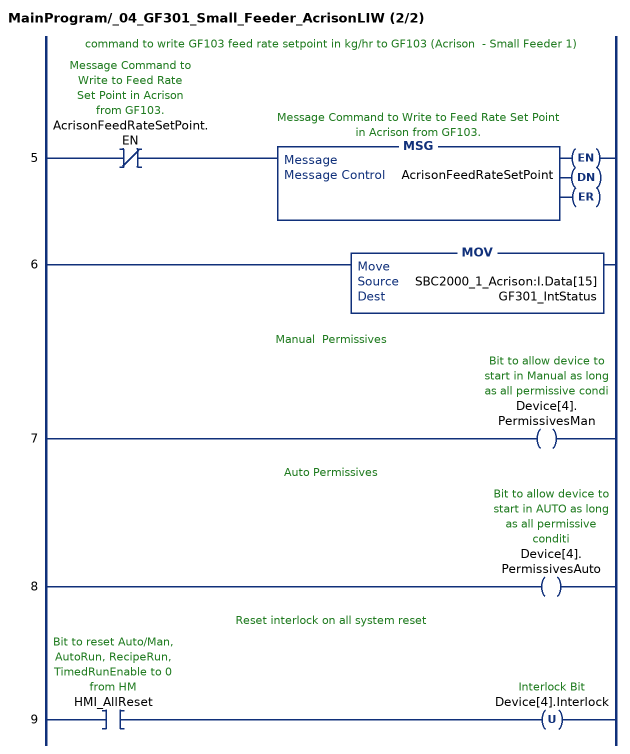
   // command to write GF103 feed rate setpoint in kg/hr to GF103 (Acrison  - Small Feeder 1)
   5: XIO(AcrisonFeedRateSetPoint.EN)MSG(AcrisonFeedRateSetPoint);
   6: MOV(SBC2000_1_Acrison:I.Data[15],GF301_IntStatus);
   // Manual  Permissives
   7: OTE(Device[4].PermissivesMan);
   // Auto Permissives
   8: OTE(Device[4].PermissivesAuto);
   // Reset interlock on all system reset
   9: XIC(HMI_AllReset)OTU(Device[4].Interlock);
END_ROUTINE

ROUTINE _05_VF101_Medium_Feeder   (* ladder *)
// Control Logix Specific to VF101 Medium Feeder
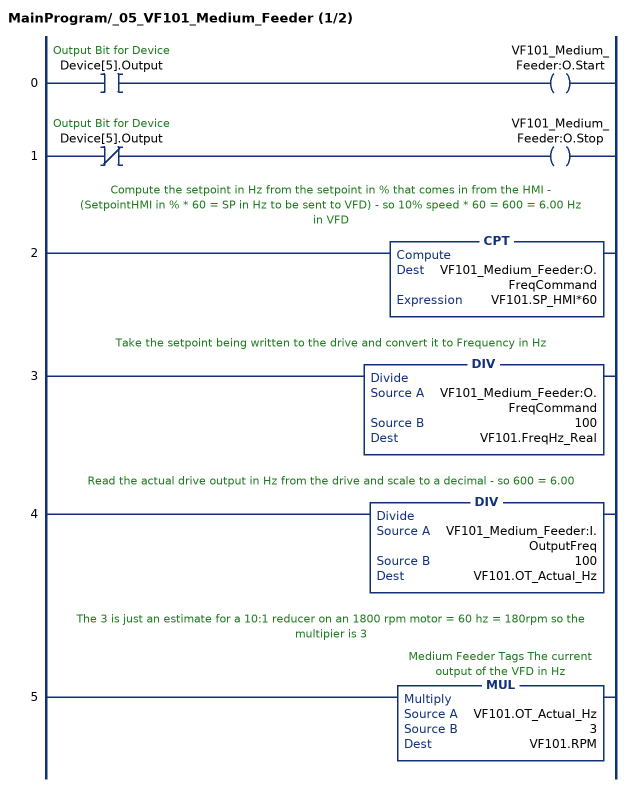
   0: XIC(Device[5].Output)OTE(VF101_Medium_Feeder:O.Start);
   1: XIO(Device[5].Output)OTE(VF101_Medium_Feeder:O.Stop);
   // Compute the setpoint in Hz from the setpoint in % that comes in from the HMI - (SetpointHMI in % * 60 = SP in Hz to be sent to VFD) - so 10% speed * 60 = 600 = 6.00 Hz in VFD
   2: CPT(VF101_Medium_Feeder:O.FreqCommand,VF101.SP_HMI*60);
   // Take the setpoint being written to the drive and convert it to Frequency in Hz
   3: DIV(VF101_Medium_Feeder:O.FreqCommand,100,VF101.FreqHz_Real);
   // Read the actual drive output in Hz from the drive and scale to a decimal - so 600 = 6.00
   4: DIV(VF101_Medium_Feeder:I.OutputFreq,100,VF101.OT_Actual_Hz);
   // The 3 is just an estimate for a 10:1 reducer on an 1800 rpm motor = 60 hz = 180rpm so the multipier is 3
   5: MUL(VF101.OT_Actual_Hz,3,VF101.RPM);
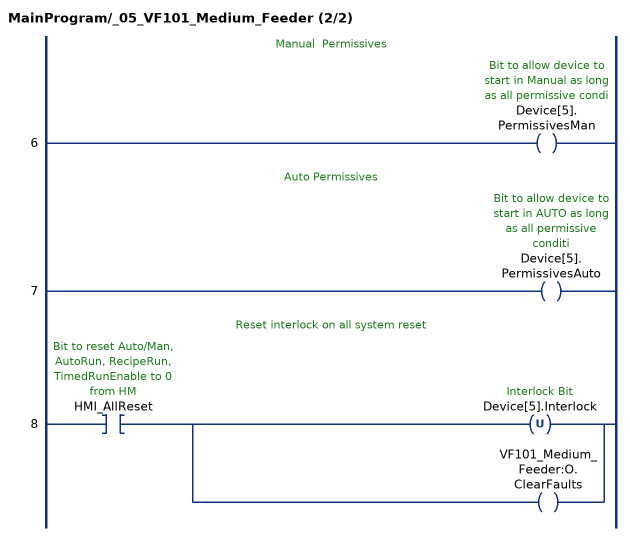
   // Manual  Permissives
   6: OTE(Device[5].PermissivesMan);
   // Auto Permissives
   7: OTE(Device[5].PermissivesAuto);
   // Reset interlock on all system reset
   8: XIC(HMI_AllReset)[OTU(Device[5].Interlock) ,OTE(VF101_Medium_Feeder:O.ClearFaults) ];
END_ROUTINE

ROUTINE _06_VF201_Small_Feeder_2   (* ladder *)
// Acison Small Feeder Control
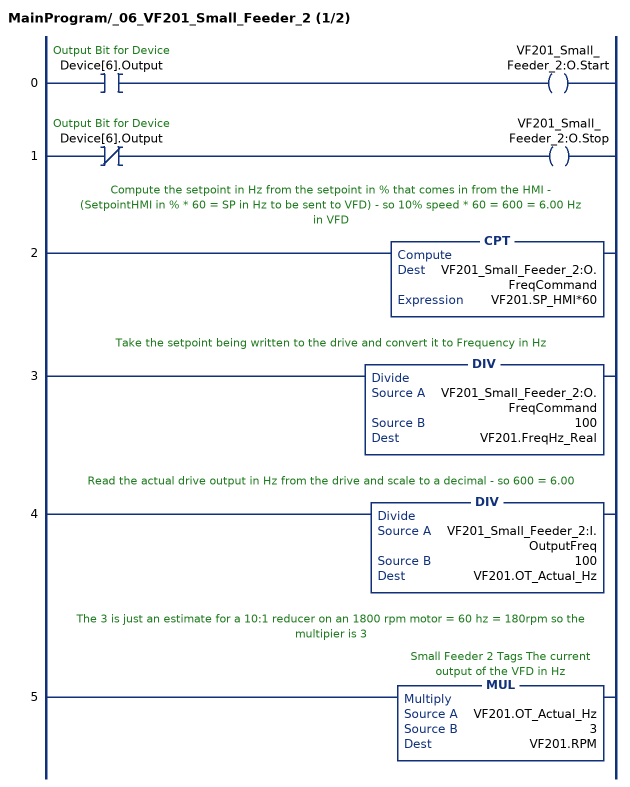
   0: XIC(Device[6].Output)OTE(VF201_Small_Feeder_2:O.Start);
   1: XIO(Device[6].Output)OTE(VF201_Small_Feeder_2:O.Stop);
   // Compute the setpoint in Hz from the setpoint in % that comes in from the HMI - (SetpointHMI in % * 60 = SP in Hz to be sent to VFD) - so 10% speed * 60 = 600 = 6.00 Hz in VFD
   2: CPT(VF201_Small_Feeder_2:O.FreqCommand,VF201.SP_HMI*60);
   // Take the setpoint being written to the drive and convert it to Frequency in Hz
   3: DIV(VF201_Small_Feeder_2:O.FreqCommand,100,VF201.FreqHz_Real);
   // Read the actual drive output in Hz from the drive and scale to a decimal - so 600 = 6.00
   4: DIV(VF201_Small_Feeder_2:I.OutputFreq,100,VF201.OT_Actual_Hz);
   // The 3 is just an estimate for a 10:1 reducer on an 1800 rpm motor = 60 hz = 180rpm so the multipier is 3
   5: MUL(VF201.OT_Actual_Hz,3,VF201.RPM);
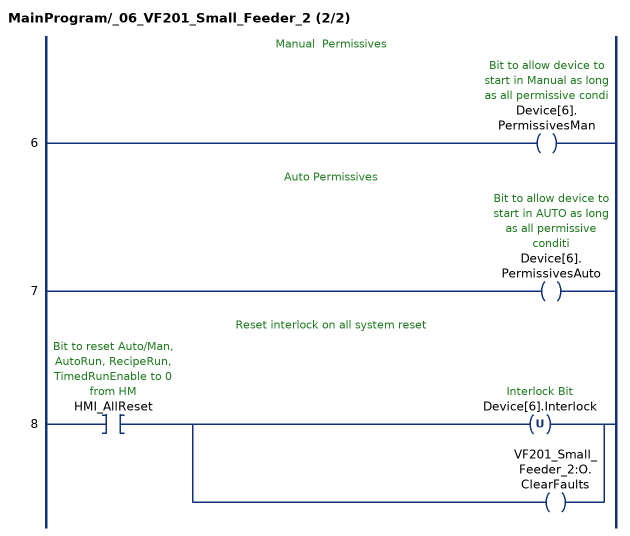
   // Manual  Permissives
   6: OTE(Device[6].PermissivesMan);
   // Auto Permissives
   7: OTE(Device[6].PermissivesAuto);
   // Reset interlock on all system reset
   8: XIC(HMI_AllReset)[OTU(Device[6].Interlock) ,OTE(VF201_Small_Feeder_2:O.ClearFaults) ];
END_ROUTINE

ROUTINE _07_FT103_Oil_Dosing   (* ladder *)
// Logic to control FT103 not associated with Device Iteration Logic
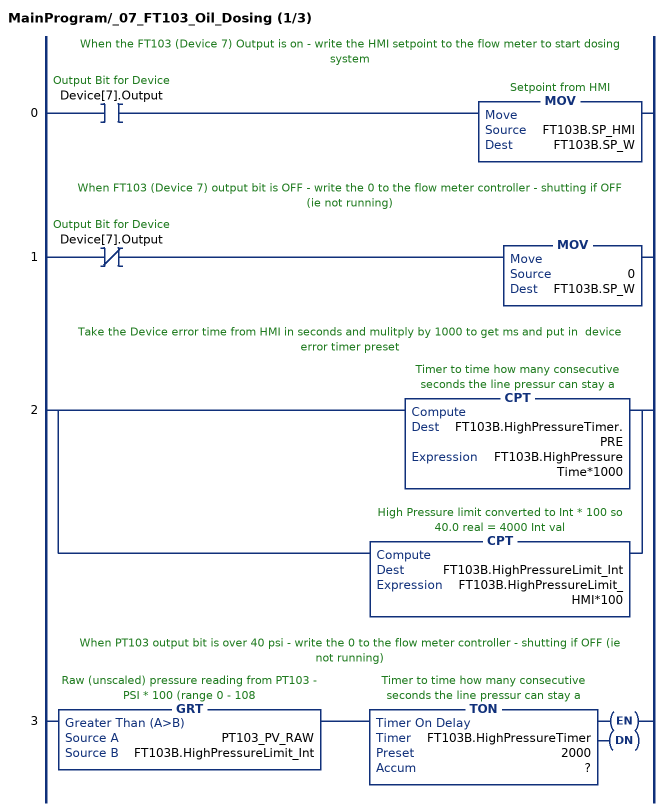
   // When the FT103 (Device 7) Output is on - write the HMI setpoint to the flow meter to start dosing system
   0: XIC(Device[7].Output)MOV(FT103B.SP_HMI,FT103B.SP_W);
   // When FT103 (Device 7) output bit is OFF - write the 0 to the flow meter controller - shutting if OFF (ie not running)
   1: XIO(Device[7].Output)MOV(0,FT103B.SP_W);
   // Take the Device error time from HMI in seconds and mulitply by 1000 to get ms and put in  device error timer preset
   2: [CPT(FT103B.HighPressureTimer.PRE,FT103B.HighPressureTime*1000) ,CPT(FT103B.HighPressureLimit_Int,FT103B.HighPressureLimit_HMI*100) ];
   // When PT103 output bit is over 40 psi - write the 0 to the flow meter controller - shutting if OFF (ie not running)
   3: GRT(PT103_PV_RAW,FT103B.HighPressureLimit_Int)TON(FT103B.HighPressureTimer,?,?);
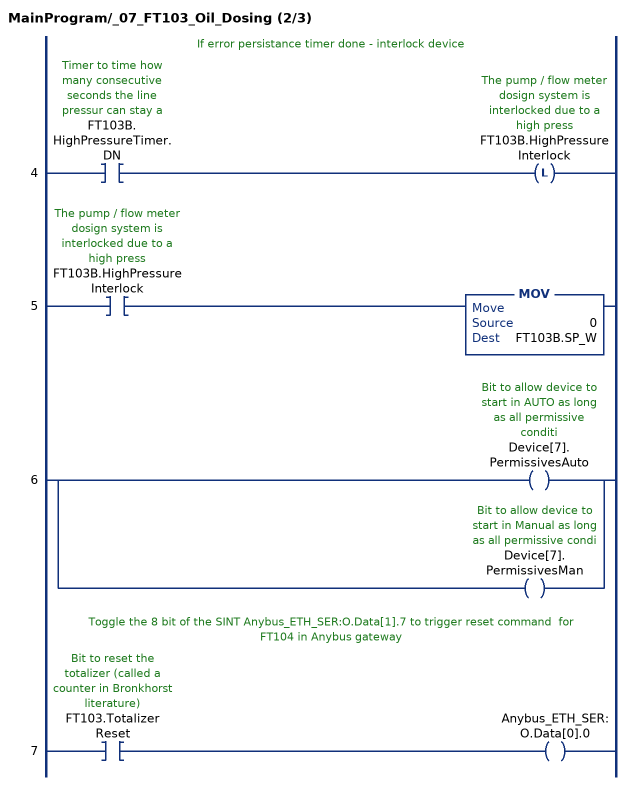
   // If error persistance timer done - interlock device
   4: XIC(FT103B.HighPressureTimer.DN)OTL(FT103B.HighPressureInterlock);
   5: XIC(FT103B.HighPressureInterlock)MOV(0,FT103B.SP_W);
   6: [OTE(Device[7].PermissivesAuto) ,OTE(Device[7].PermissivesMan) ];
   // Toggle the 8 bit of the SINT Anybus_ETH_SER:O.Data[1].7 to trigger reset command  for FT104 in Anybus gateway
   7: XIC(FT103.TotalizerReset)OTE(Anybus_ETH_SER:O.Data[0].0);
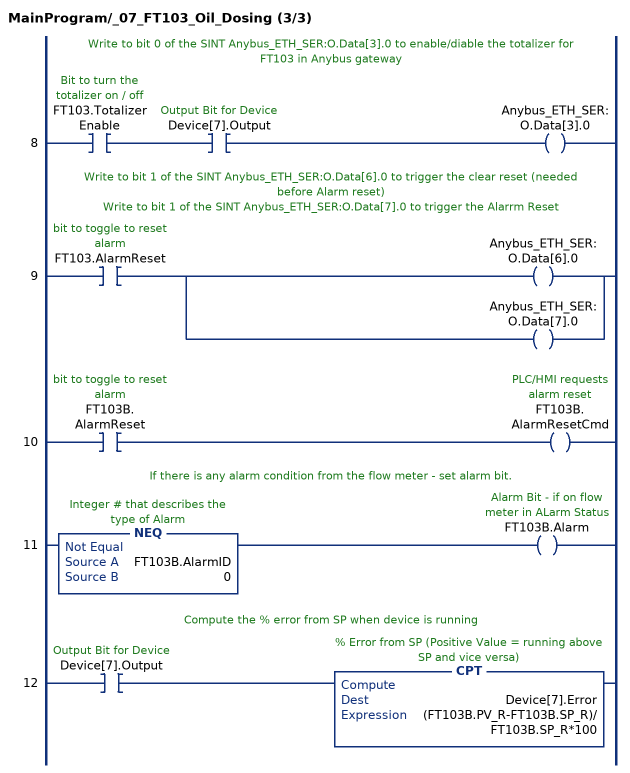
   // Write to bit 0 of the SINT Anybus_ETH_SER:O.Data[3].0 to enable/diable the totalizer for FT103 in Anybus gateway
   8: XIC(FT103.TotalizerEnable)XIC(Device[7].Output)OTE(Anybus_ETH_SER:O.Data[3].0);
   // Write to bit 1 of the SINT Anybus_ETH_SER:O.Data[6].0 to trigger the clear reset (needed before Alarm reset)
   // Write to bit 1 of the SINT Anybus_ETH_SER:O.Data[7].0 to trigger the Alarrm Reset
   9: XIC(FT103.AlarmReset)[OTE(Anybus_ETH_SER:O.Data[6].0) ,OTE(Anybus_ETH_SER:O.Data[7].0) ];
   10: XIC(FT103B.AlarmReset)OTE(FT103B.AlarmResetCmd);
   // If there is any alarm condition from the flow meter - set alarm bit.
   11: NEQ(FT103B.AlarmID,0)OTE(FT103B.Alarm);
   // Compute the % error from SP when device is running
   12: XIC(Device[7].Output)CPT(Device[7].Error,(FT103B.PV_R-FT103B.SP_R)/FT103B.SP_R*100);
END_ROUTINE
